# EPICS substitutions: iocs/BL11I-EA-IOC-12/BL11I-EA-IOC-12App/Db/BL11I-EA-IOC-12_expanded.substitutions
# This file was automatically generated on Tue 29 Sep 2026 10:59:15 BST from
# source: /scratch/djp75990/code/I11/bl11i-builder/etc/makeIocs/BL11I-EA-IOC-12.xml
#
# *** Please do not edit this file: edit the source file instead. ***
#

# Macros:
#  IOC  Device prefix
file $(DEVIOCSTATS)/db/iocAdminSoft.db
{
pattern { IOC }
    { "BL11I-EA-IOC-12" }
}

# Macros:
#  IOC  Device prefix
file $(DEVIOCSTATS)/db/iocAdminScanMon.db
{
pattern { IOC }
    { "BL11I-EA-IOC-12" }
}

# Macros:
#  name      name for gui elements
#  EDM_FILE  edm screen, defaults to ioc_stats_softdls.edl
#  IOC       ioc name
file $(DEVIOCSTATS)/db/iocGui.db
{
pattern { name, EDM_FILE, IOC }
    { "EA12_STATS", "ioc_stats_softdls.edl", "BL11I-EA-IOC-12" }
}

# Macros:
#  P     Template argument
#  Q     Template argument
#  PORT  Template argument
#  UID   Template argument
file $(OXINSTCRYOJET)/db/MercuryiTC-SCPI_heater.template
{
pattern { P, Q, PORT, UID }
    { "BL11I-EA-TEMPC-03", ":MERC", "ITC_CTLR", "MB0.H1" }
}

# Macros:
#  P     Template argument
#  Q     Template argument
#  PORT  Template argument
#  UID   Template argument
file $(OXINSTCRYOJET)/db/MercuryiTC-SCPI_loop.template
{
pattern { P, Q, PORT, UID }
    { "BL11I-EA-TEMPC-03", ":MERC", "ITC_CTLR", "MB1.T1" }
}

# Macros:
#  P     Template argument
#  Q     Template argument
#  PORT  Template argument
file $(OXINSTCRYOJET)/db/MercuryiTC-SCPI_system.template
{
pattern { P, Q, PORT }
    { "BL11I-EA-TEMPC-03", ":MERC", "ITC_CTLR" }
}

# Macros:
#  P     Template argument
#  Q     Template argument
#  PORT  Template argument
#  UID   Template argument
file $(OXINSTCRYOJET)/db/MercuryiTC-SCPI_tempSensor.template
{
pattern { P, Q, PORT, UID }
    { "BL11I-EA-TEMPC-03", ":MERC", "ITC_CTLR", "MB1.T1" }
}
